(* Logix 5000 project; controller furnace vendor 1 type 14 code 92 rev 32.11; software revision 32.00 *)

TASK MainTask (continuous, watchdog 500 ms) : MainProgram

MODULES
   Local : vendor 1 type 14 code 92 (ICP 0, rev 32.11)
      inputfurnace : 1756-IB32 (ICP 1, rev 2.1, Input RPI 20 ms)
      outputfurnace : vendor 1 type 7 code 8 (ICP 2, rev 1.1, Output RPI 20 ms)
      ANYTHING : 1756-IF8 (ICP 3, rev 1.1, Input RPI 100 ms)
END_MODULES

VAR_GLOBAL   (* controller tags *)
   COLD_END_TEMP : ALIAS FOR Local:3:I.Ch1Data;   // Cold end temperature
   ENTR_CONV_ON : ALIAS FOR Local:2:O.Data.13;   // Entrance conveyor control
   ENTR_DOOR_LS : ALIAS FOR Local:1:I.Data.17;   // Plate at furnace entrance limit switch
   ENTR_DOOR_PROX : ALIAS FOR Local:1:I.Data.18;   // Entrance door optical thru sensor
   ENTR_HORIZ_ELS : ALIAS FOR Local:1:I.Data.5;   // Entrance horiz cylinder extended limit switch
   ENTR_HORIZ_EXT : ALIAS FOR Local:2:O.Data.10;   // Entrance horizontal extend control
   ENTR_HORIZ_RET : ALIAS FOR Local:2:O.Data.9;   // Entrance horizontal retract control
   ENTR_HORIZ_RLS : ALIAS FOR Local:1:I.Data.4;   // Entrance horiz cylinder retracted limit switch
   ENTR_PLAT_IN_PROX : ALIAS FOR Local:1:I.Data.16;   // Entrance conveyor plate in prox switch
   EXIT_CONV_ON : ALIAS FOR Local:2:O.Data.14;   // Exit conveyor control
   EXIT_DOOR_DOWN : ALIAS FOR Local:2:O.Data.7;   // Exit door down control
   EXIT_DOOR_LF_DLS : ALIAS FOR Local:1:I.Data.14;   // Exit door left side down limit switch
   EXIT_DOOR_LF_ULS : ALIAS FOR Local:1:I.Data.13;   // Exit door left side up limit switch
   EXIT_DOOR_PROX : ALIAS FOR Local:1:I.Data.19;   // Exit door optical thru sensor
   EXIT_DOOR_RG_DLS : ALIAS FOR Local:1:I.Data.12;   // Exit door right side down limit switch
   EXIT_DOOR_RG_ULS : ALIAS FOR Local:1:I.Data.11;   // Exit door right side up limit switch
   EXIT_DOOR_UP : ALIAS FOR Local:2:O.Data.8;   // Exit door up control
   EXIT_HORIZ_ELS : ALIAS FOR Local:1:I.Data.7;   // Exit horiz fork cylinder extended limit switch
   EXIT_HORIZ_EXT : ALIAS FOR Local:2:O.Data.6;   // Exit fork horizontal extend control
   EXIT_HORIZ_RET : ALIAS FOR Local:2:O.Data.5;   // Exit fork horizontal retract control
   EXIT_HORIZ_RLS : ALIAS FOR Local:1:I.Data.6;   // Exit horiz fork cylinder retracted limit switch
   EXIT_PLAT_OUT_PROX : ALIAS FOR Local:1:I.Data.15;   // Exit conveyor plate out prox switch
   EXIT_VERT_DLS : ALIAS FOR Local:1:I.Data.8;   // Exit vertical fork cylinder down limit switch
   EXIT_VERT_DOWN : ALIAS FOR Local:2:O.Data.3;   // Exit fork vertical down control
   EXIT_VERT_MLS : ALIAS FOR Local:1:I.Data.9;   // Exit vertical fork cylinder middle limit switch
   EXIT_VERT_ULS : ALIAS FOR Local:1:I.Data.10;   // Exit vertical fork cylinder up limit switch
   EXIT_VERT_UP : ALIAS FOR Local:2:O.Data.4;   // Exit fork vertical up control
   HEATER_ON : ALIAS FOR Local:2:O.Data.15;   // Furnace heater control
   HOT_END_TEMP : ALIAS FOR Local:3:I.Ch0Data;   // Hot end temperature
   RESET_SW : ALIAS FOR Local:1:I.Data.2;   // Reset pushbutton
   RStep_1 : BOOL;
   RStep_10 : BOOL;
   RStep_11 : BOOL;
   RStep_12 : BOOL;
   RStep_13 : BOOL;
   RStep_14 : BOOL;
   RStep_15 : BOOL;
   RStep_16 : BOOL;
   RStep_17 : BOOL;
   RStep_18 : BOOL;
   RStep_19 : BOOL;
   RStep_2 : BOOL;
   RStep_3 : BOOL;
   RStep_4 : BOOL;
   RStep_5 : BOOL;
   RStep_6 : BOOL;
   RStep_7 : BOOL;
   RStep_8 : BOOL;
   RStep_9 : BOOL;
   RUN_LA : ALIAS FOR Local:2:O.Data.0;   // ON when operation is running
   START_PB : ALIAS FOR Local:1:I.Data.0;   // Start pushbutton
   Step_1 : BOOL;
   Step_10 : BOOL;
   Step_11 : BOOL;
   Step_12 : BOOL;
   Step_13 : BOOL := 1;
   Step_14 : BOOL;
   Step_15 : BOOL;
   Step_16 : BOOL;
   Step_17 : BOOL;
   Step_18 : BOOL;
   Step_19 : BOOL;
   Step_2 : BOOL;
   Step_20 : BOOL;
   Step_21 : BOOL;
   Step_22 : BOOL;
   Step_23 : BOOL;
   Step_24 : BOOL;
   Step_25 : BOOL;
   Step_26 : BOOL;
   Step_27 : BOOL;
   Step_28 : BOOL;
   Step_29 : BOOL;
   Step_3 : BOOL;
   Step_30 : BOOL;
   Step_31 : BOOL;
   Step_32 : BOOL;
   Step_33 : BOOL;
   Step_34 : BOOL;
   Step_35 : BOOL;
   Step_36 : BOOL;
   Step_37 : BOOL;
   Step_38 : BOOL;
   Step_39 : BOOL;
   Step_4 : BOOL;
   Step_40 : BOOL;
   Step_41 : BOOL;
   Step_42 : BOOL;
   Step_43 : BOOL;
   Step_44 : BOOL;
   Step_45 : BOOL;
   Step_46 : BOOL;
   Step_47 : BOOL;
   Step_48 : BOOL;
   Step_49 : BOOL;
   Step_5 : BOOL;
   Step_50 : BOOL;
   Step_51 : BOOL;
   Step_52 : BOOL;
   Step_53 : BOOL;
   Step_54 : BOOL;
   Step_55 : BOOL;
   Step_6 : BOOL;
   Step_7 : BOOL;
   Step_8 : BOOL;
   Step_9 : BOOL;
   STOP_PB : ALIAS FOR Local:1:I.Data.1;   // Stop pushbutton
END_VAR

PROGRAM MainProgram   (* main routine MainRoutine *)
VAR
   HOTCONV : DINT;
   Int_Reset : BOOL;
   RUN : BOOL;
   TMR1 : TIMER := (PRE := 10000);
   TMR2 : TIMER := (PRE := 10000);
   tmr3 : TIMER := (PRE := 15000);
   TMR4 : TIMER := (PRE := 5000);
END_VAR

ROUTINE MainRoutine   (* ladder *)
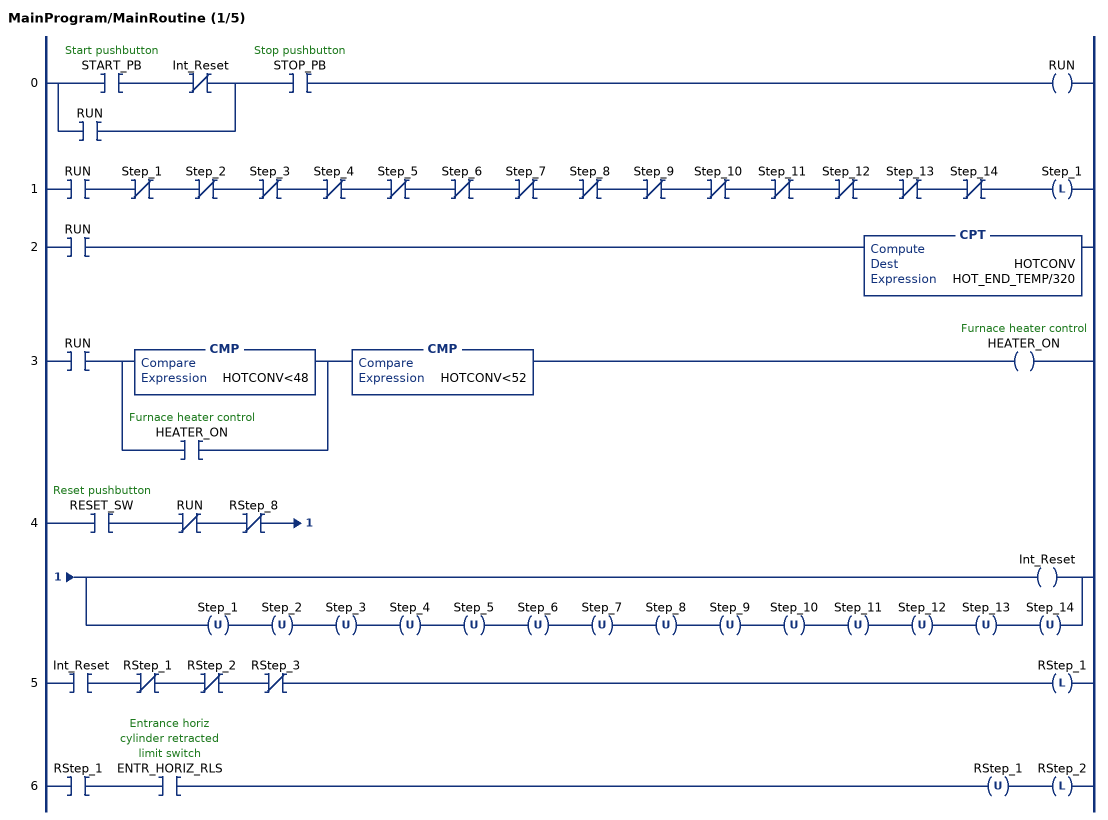
   0: [XIC(START_PB) XIO(Int_Reset) ,XIC(RUN) ]XIC(STOP_PB)OTE(RUN);
   1: XIC(RUN)XIO(Step_1)XIO(Step_2)XIO(Step_3)XIO(Step_4)XIO(Step_5)XIO(Step_6)XIO(Step_7)XIO(Step_8)XIO(Step_9)XIO(Step_10)XIO(Step_11)XIO(Step_12)XIO(Step_13)XIO(Step_14)OTL(Step_1);
   2: XIC(RUN)CPT(HOTCONV,HOT_END_TEMP/320);
   3: XIC(RUN)[CMP(HOTCONV<48) ,XIC(HEATER_ON) ]CMP(HOTCONV<52)OTE(HEATER_ON);
   4: XIC(RESET_SW)XIO(RUN)XIO(RStep_8)[OTE(Int_Reset) ,OTU(Step_1) OTU(Step_2) OTU(Step_3) OTU(Step_4) OTU(Step_5) OTU(Step_6) OTU(Step_7) OTU(Step_8) OTU(Step_9) OTU(Step_10) OTU(Step_11) OTU(Step_12) OTU(Step_13) OTU(Step_14) ];
   5: XIC(Int_Reset)XIO(RStep_1)XIO(RStep_2)XIO(RStep_3)OTL(RStep_1);
   6: XIC(RStep_1)XIC(ENTR_HORIZ_RLS)OTU(RStep_1)OTL(RStep_2);
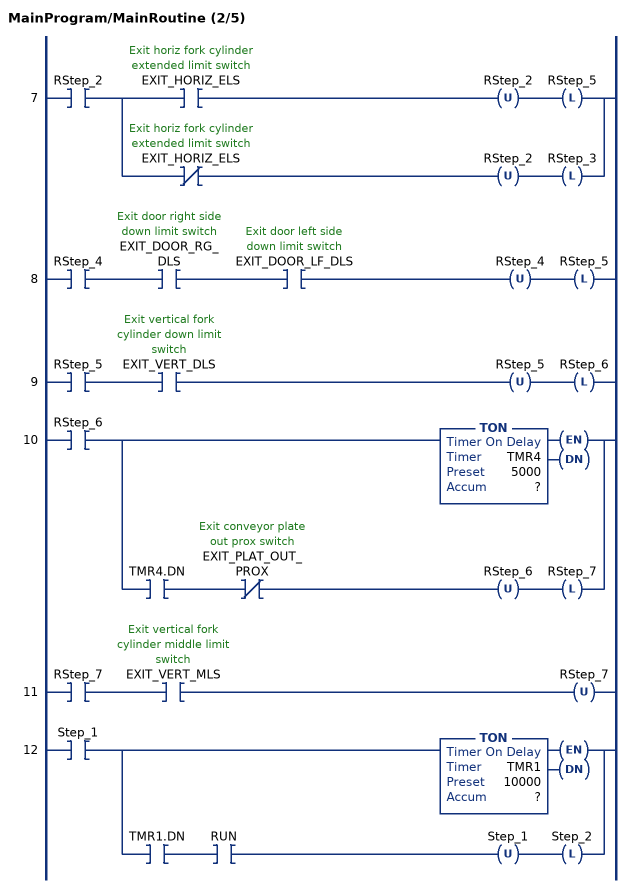
   7: XIC(RStep_2)[XIC(EXIT_HORIZ_ELS) OTU(RStep_2) OTL(RStep_5) ,XIO(EXIT_HORIZ_ELS) OTU(RStep_2) OTL(RStep_3) ];
   8: XIC(RStep_4)XIC(EXIT_DOOR_RG_DLS)XIC(EXIT_DOOR_LF_DLS)OTU(RStep_4)OTL(RStep_5);
   9: XIC(RStep_5)XIC(EXIT_VERT_DLS)OTU(RStep_5)OTL(RStep_6);
   10: XIC(RStep_6)[TON(TMR4,?,?) ,XIC(TMR4.DN) XIO(EXIT_PLAT_OUT_PROX) OTU(RStep_6) OTL(RStep_7) ];
   11: XIC(RStep_7)XIC(EXIT_VERT_MLS)OTU(RStep_7);
   12: XIC(Step_1)[TON(TMR1,?,?) ,XIC(TMR1.DN) XIC(RUN) OTU(Step_1) OTL(Step_2) ];
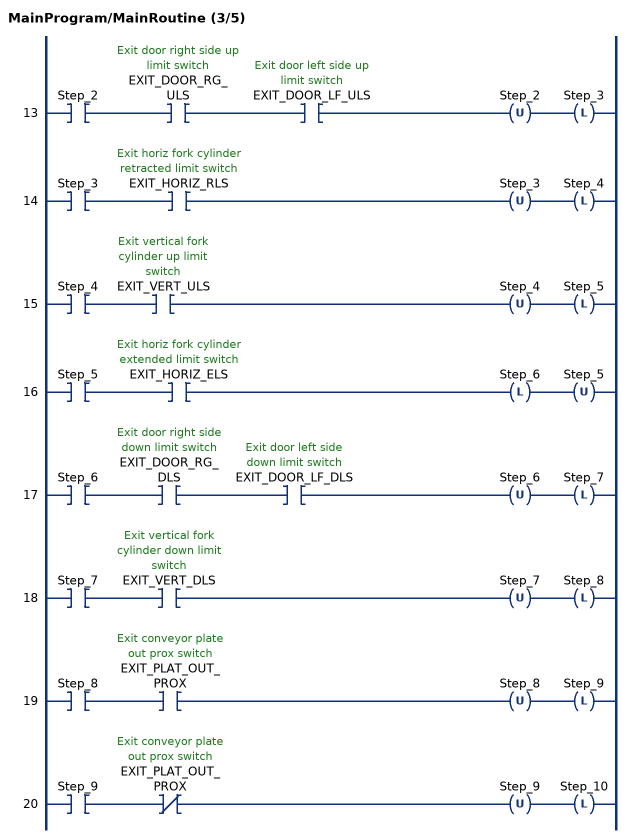
   13: XIC(Step_2)XIC(EXIT_DOOR_RG_ULS)XIC(EXIT_DOOR_LF_ULS)OTU(Step_2)OTL(Step_3);
   14: XIC(Step_3)XIC(EXIT_HORIZ_RLS)OTU(Step_3)OTL(Step_4);
   15: XIC(Step_4)XIC(EXIT_VERT_ULS)OTU(Step_4)OTL(Step_5);
   16: XIC(Step_5)XIC(EXIT_HORIZ_ELS)OTL(Step_6)OTU(Step_5);
   17: XIC(Step_6)XIC(EXIT_DOOR_RG_DLS)XIC(EXIT_DOOR_LF_DLS)OTU(Step_6)OTL(Step_7);
   18: XIC(Step_7)XIC(EXIT_VERT_DLS)OTU(Step_7)OTL(Step_8);
   19: XIC(Step_8)XIC(EXIT_PLAT_OUT_PROX)OTU(Step_8)OTL(Step_9);
   20: XIC(Step_9)XIO(EXIT_PLAT_OUT_PROX)OTU(Step_9)OTL(Step_10);
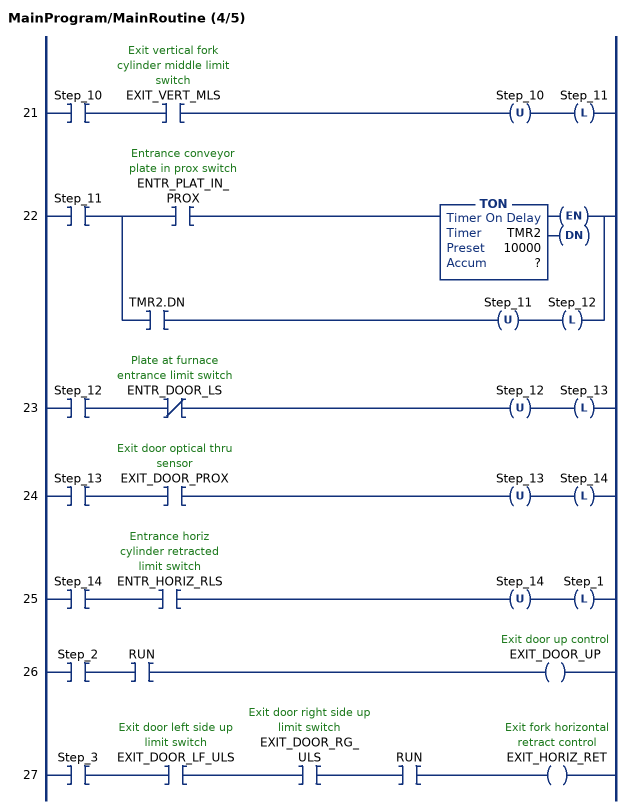
   21: XIC(Step_10)XIC(EXIT_VERT_MLS)OTU(Step_10)OTL(Step_11);
   22: XIC(Step_11)[XIC(ENTR_PLAT_IN_PROX) TON(TMR2,?,?) ,XIC(TMR2.DN) OTU(Step_11) OTL(Step_12) ];
   23: XIC(Step_12)XIO(ENTR_DOOR_LS)OTU(Step_12)OTL(Step_13);
   24: XIC(Step_13)XIC(EXIT_DOOR_PROX)OTU(Step_13)OTL(Step_14);
   25: XIC(Step_14)XIC(ENTR_HORIZ_RLS)OTU(Step_14)OTL(Step_1);
   26: XIC(Step_2)XIC(RUN)OTE(EXIT_DOOR_UP);
   27: XIC(Step_3)XIC(EXIT_DOOR_LF_ULS)XIC(EXIT_DOOR_RG_ULS)XIC(RUN)OTE(EXIT_HORIZ_RET);
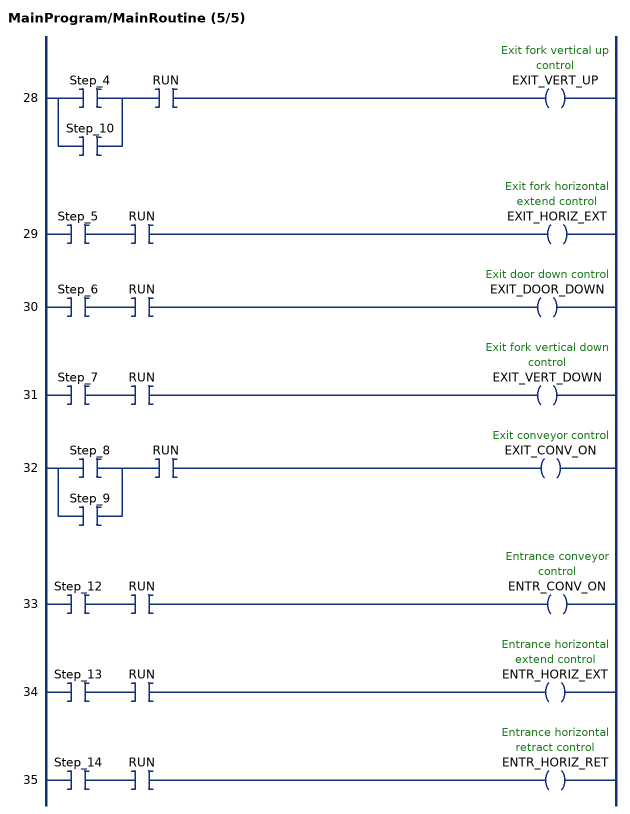
   28: [XIC(Step_4) ,XIC(Step_10) ]XIC(RUN)OTE(EXIT_VERT_UP);
   29: XIC(Step_5)XIC(RUN)OTE(EXIT_HORIZ_EXT);
   30: XIC(Step_6)XIC(RUN)OTE(EXIT_DOOR_DOWN);
   31: XIC(Step_7)XIC(RUN)OTE(EXIT_VERT_DOWN);
   32: [XIC(Step_8) ,XIC(Step_9) ]XIC(RUN)OTE(EXIT_CONV_ON);
   33: XIC(Step_12)XIC(RUN)OTE(ENTR_CONV_ON);
   34: XIC(Step_13)XIC(RUN)OTE(ENTR_HORIZ_EXT);
   35: XIC(Step_14)XIC(RUN)OTE(ENTR_HORIZ_RET);
END_ROUTINE
END_PROGRAM
